# EPICS substitutions: scllrfApp/Db/RESRegisters.substitutions
file scllrfRES.template
{
	{ NULL = NULL }
}

file scllrfCommon.template
{
	{ NULL = NULL }
}
